FUNCTION_BLOCK SUB (* Subtract *)
  (* Standard: 61499-2 *)
  (* Version 1.0, 02.01.2011, gsha041, UoA, Initial Version *)
  (* Compiler header: package fb.rt.UoA; *)
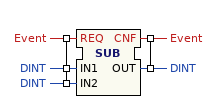
  EVENT_INPUT
    REQ WITH IN1, IN2; (* Normal Execution Request *)
  END_EVENT
  EVENT_OUTPUT
    CNF WITH OUT; (* Execution Confirmation *)
  END_EVENT
  VAR_INPUT
    IN1 : DINT; (* Argument *)
    IN2 : DINT; (* Argument *)
  END_VAR
  VAR_OUTPUT
    OUT : DINT; (* Result: IN1 - IN2 - IN3 - ... *)
  END_VAR
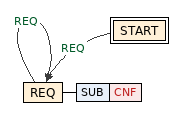
  EC_STATES
    START; (* Initial State *)
    REQ : SUB -> CNF; (* Normal execution *)
  END_STATES
  EC_TRANSITIONS
    START TO REQ := REQ;
    REQ TO REQ := REQ;
  END_TRANSITIONS
  ALGORITHM SUB IN ST: (* Normally executed algorithm *)
OUT := IN1 - IN2;
  END_ALGORITHM
END_FUNCTION_BLOCK
